{attribute 'qualified_only'}
{attribute 'strict'}
TYPE TmsSwitchMode :
(
	Automatic := 0,
	Manual := 1
);
END_TYPE

(* stored: Version 1.1.0.1, ProductVersion 3.1.4024.11
   DUT TmsSwitchMode: Id {2d21ed61-d148-4fc6-849d-4a38d246d8dd} *)
